# EPICS substitutions: iocBoot/iocTml/singleAxis.substitutions
file "$(TOP)/db/motor.db"
{
    pattern
    { P,      M,    DESC,            PORT,  ADDR, MRES, ARES, EGU,    DHLM,    DLLM,   VELO, ACCS, TWV }
    { "TEST:MOT:TML:", "TESTFLG", "TML Axis 0",   "TML1", 0,   1.0,  1.0,  "ustep", 100000, -100000, 15,   0.5,  100  }
}
